TYPE DriveReference :
STRUCT
	drive : REFERENCE TO IntegratedDrive;
END_STRUCT
END_TYPE

(* stored: Version 1.1.0.1, ProductVersion 3.1.4024.2
   DUT DriveReference: Id {9dea8eff-8799-4ed8-8d12-e74b667616f8} *)
